// Mitsubishi GX Works2 project: PLCmaymay1kim   PLC: FX3U/FX3UC

PROGRAM MAIN
VAR
  Y008 : BOOL;
END_VAR
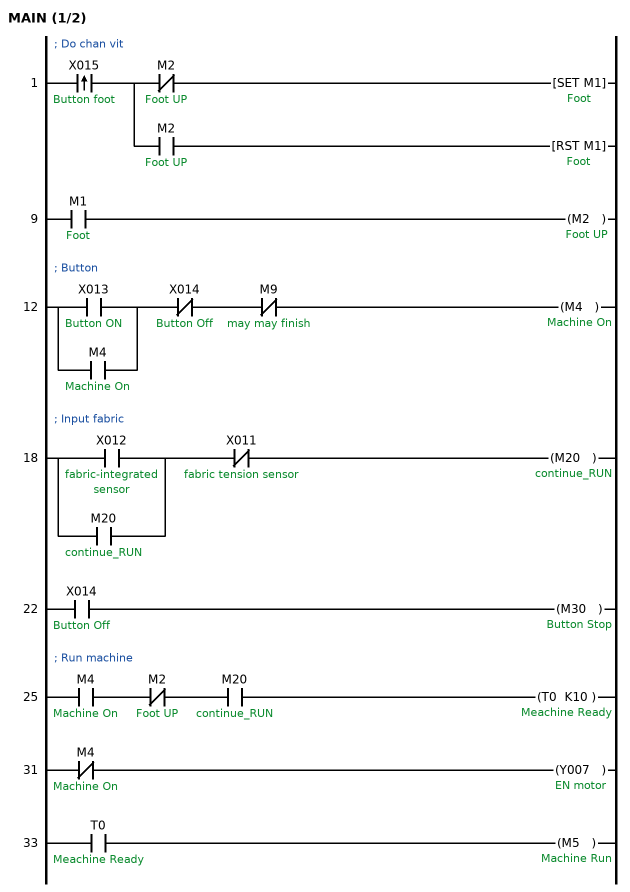
; Do chan vit
1     LDP     X015  ; Button foot
      MPS
      ANI     M2  ; Foot UP
      SET     M1  ; Foot
      MPP
      AND     M2  ; Foot UP
      RST     M1  ; Foot
9     LD      M1  ; Foot
      OUT     M2  ; Foot UP
; Button
12    LD      X013  ; Button ON
      OR      M4  ; Machine On
      ANI     X014  ; Button Off
      ANI     M9  ; may may finish
      OUT     M4  ; Machine On
; Input fabric
18    LD      X012  ; fabric-integrated sensor
      OR      M20  ; continue_RUN
      ANI     X011  ; fabric tension sensor
      OUT     M20  ; continue_RUN
22    LD      X014  ; Button Off
      OUT     M30  ; Button Stop
; Run machine
25    LD      M4  ; Machine On
      ANI     M2  ; Foot UP
      AND     M20  ; continue_RUN
      OUT     T0 K10  ; Meachine Ready
31    LDI     M4  ; Machine On
      OUT     Y007  ; EN motor
33    LD      T0  ; Meachine Ready
      OUT     M5  ; Machine Run
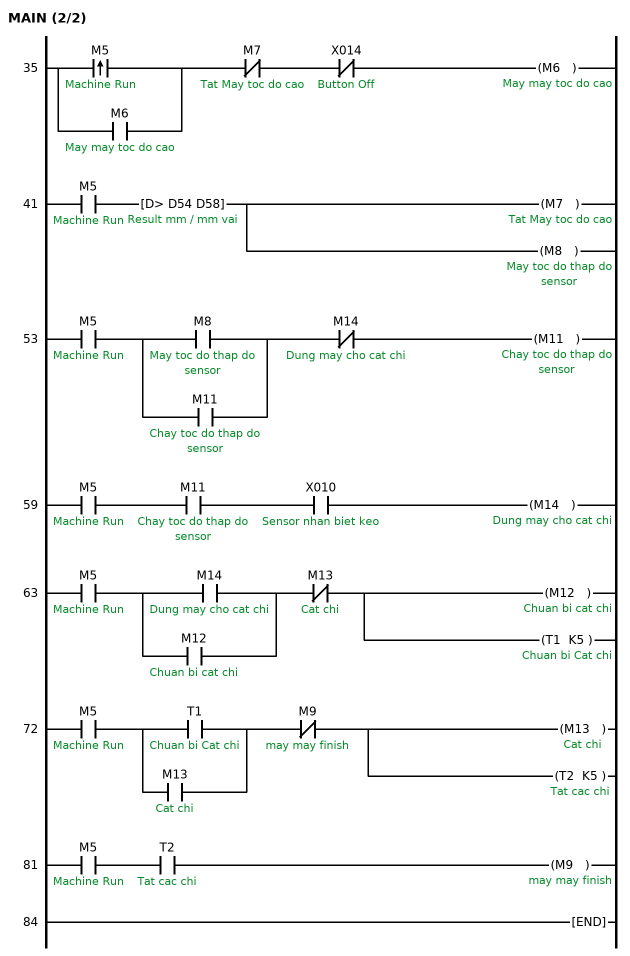
35    LDP     M5  ; Machine Run
      OR      M6  ; May may toc do cao
      ANI     M7  ; Tat May toc do cao
      ANI     X014  ; Button Off
      OUT     M6  ; May may toc do cao
41    LD      M5  ; Machine Run
      ANDD>   D54 D58  ; Result mm / mm vai
      OUT     M7  ; Tat May toc do cao
      OUT     M8  ; May toc do thap do sensor
53    LD      M5  ; Machine Run
      LD      M8  ; May toc do thap do sensor
      OR      M11  ; Chay toc do thap do sensor
      ANB
      ANI     M14  ; Dung may cho cat chi
      OUT     M11  ; Chay toc do thap do sensor
59    LD      M5  ; Machine Run
      AND     M11  ; Chay toc do thap do sensor
      AND     X010  ; Sensor nhan biet keo
      OUT     M14  ; Dung may cho cat chi
63    LD      M5  ; Machine Run
      LD      M14  ; Dung may cho cat chi
      OR      M12  ; Chuan bi cat chi
      ANB
      ANI     M13  ; Cat chi
      OUT     M12  ; Chuan bi cat chi
      OUT     T1 K5  ; Chuan bi Cat chi
72    LD      M5  ; Machine Run
      LD      T1  ; Chuan bi Cat chi
      OR      M13  ; Cat chi
      ANB
      ANI     M9  ; may may finish
      OUT     M13  ; Cat chi
      OUT     T2 K5  ; Tat cac chi
81    LD      M5  ; Machine Run
      AND     T2  ; Tat cac chi
      OUT     M9  ; may may finish
84    END
END_PROGRAM

PROGRAM OUTPUT
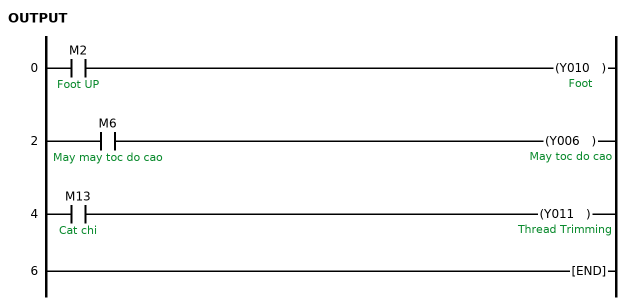
0     LD      M2  ; Foot UP
      OUT     Y010  ; Foot
2     LD      M6  ; May may toc do cao
      OUT     Y006  ; May toc do cao
4     LD      M13  ; Cat chi
      OUT     Y011  ; Thread Trimming
6     END
END_PROGRAM

PROGRAM Sewing
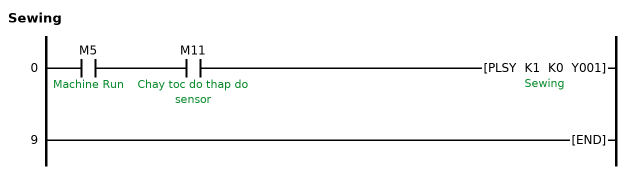
0     LD      M5  ; Machine Run
      AND     M11  ; Chay toc do thap do sensor
      PLSY    K1 K0 Y001  ; Sewing
9     END
END_PROGRAM

PROGRAM Motor
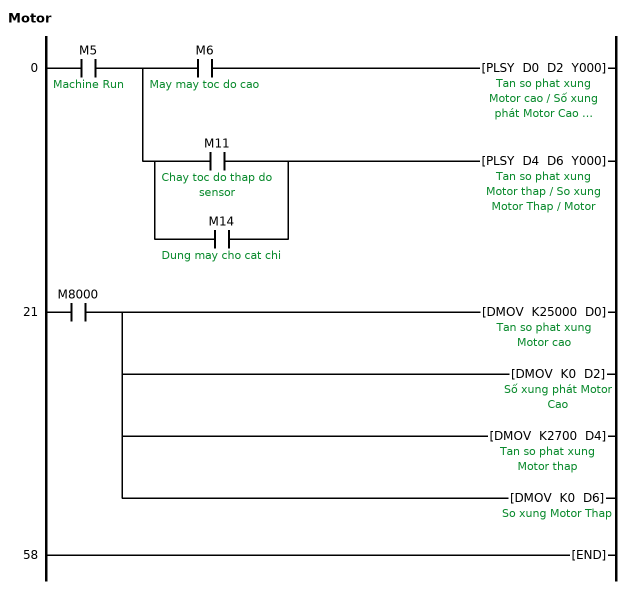
0     LD      M5  ; Machine Run
      MPS
      AND     M6  ; May may toc do cao
      PLSY    D0 D2 Y000  ; Tan so phat xung Motor cao / Số xung phát Motor Cao / Motor
      MPP
      LD      M11  ; Chay toc do thap do sensor
      OR      M14  ; Dung may cho cat chi
      ANB
      PLSY    D4 D6 Y000  ; Tan so phat xung Motor thap / So xung Motor Thap / Motor
21    LD      M8000
      DMOV    K25000 D0
      DMOV    K0 D2
      DMOV    K2700 D4
      DMOV    K0 D6
58    END
END_PROGRAM

PROGRAM Meter_En
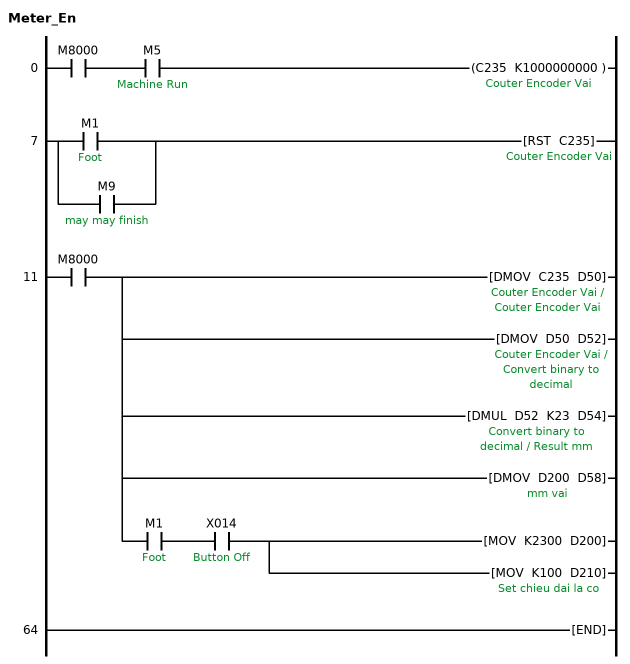
0     LD      M8000
      AND     M5  ; Machine Run
      OUT     C235 K1000000000  ; Couter Encoder Vai
7     LD      M1  ; Foot
      OR      M9  ; may may finish
      RST     C235  ; Couter Encoder Vai
11    LD      M8000
      DMOV    C235 D50  ; Couter Encoder Vai
      DMOV    D50 D52  ; Convert binary to decimal
      DMUL    D52 K23 D54  ; Result mm
      DMOV    D200 D58  ; mm vai
      AND     M1  ; Foot
      AND     X014  ; Button Off
      MOV     K2300 D200
      MOV     K100 D210  ; Set chieu dai la co
64    END
END_PROGRAM

PROGRAM Thread
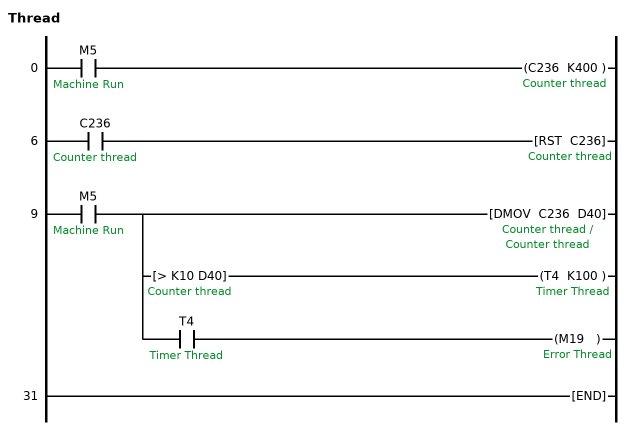
0     LD      M5  ; Machine Run
      OUT     C236 K400  ; Counter thread
6     LD      C236  ; Counter thread
      RST     C236  ; Counter thread
9     LD      M5  ; Machine Run
      DMOV    C236 D40  ; Counter thread
      MPS
      AND>    K10 D40  ; Counter thread
      OUT     T4 K100  ; Timer Thread
      MPP
      AND     T4  ; Timer Thread
      OUT     M19  ; Error Thread
31    END
END_PROGRAM

PROGRAM MODBUS
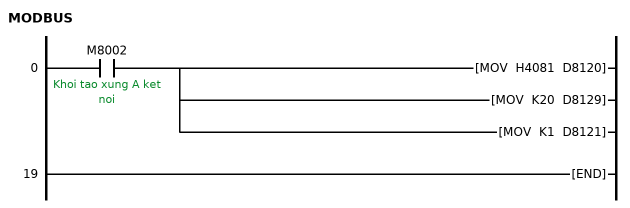
0     LD      M8002  ; Khoi tao xung A ket noi
      MOV     H4081 D8120
        [note] Modbus RTU, 9600, ODD, 8
      MOV     K20 D8129
        [note] Timeout
      MOV     K1 D8121
        [note] Station Slave = 1
19    END
END_PROGRAM

// device comments not shown above
X000  ; Sensor vong quay may may
M3  ; Foot down
M15  ; Chay dem xung la co
M16  ; Chay du so xung thi dung
M17  ; Chay du so xung thi dung
M18  ; Chay lai bat sensor
T3  ; Chay xung con lai
D10  ; So xung cua chieu dai la co
D12  ; So xung chay den keo
D14  ; Thoi gian tang giam Motor
D20  ; chieu dai la co
D22  ; So xung phat sewing
D24  ; thoi gian tang giam sewing
D30  ; Tan so phat xung Motor
D32  ; So xung phat Motot
D34  ; Thoi gian tang giam Motor
D56  ; mmx100
C0  ; Dem so xung cua mieng vai
